// TwinCAT 3 PLC project ClassDemo
// ProgramVersion: 3.1.4023.0
// libraries:
//   Tc2_Standard, * (Beckhoff Automation GmbH)
//   Tc2_System, * (Beckhoff Automation GmbH)
//   Tc3_Module, * (Beckhoff Automation GmbH)
// project tree:
//   / PlcTask.TcTTO (not stored)
//   POUs/ MAIN.TcPOU, Motor.TcPOU (not stored), Plc_Prog.TcPOU (not stored)

// ---- POUs/MAIN.TcPOU
PROGRAM MAIN
VAR
END_VAR

Plc_Prog();

END_PROGRAM
